# EPICS substitutions: opcpaepsApp/Db/eps_chiller_loop.substitutions
file eps_chiller_loop.template {
  pattern
    {ID}
    {"01"}
    {"02"}
    {"03"}
    {"04"}
}
